// TIA Portal V17 export
// export: Created 2024-09-02T12:50:30.4708578Z, ExportSetting WithDefaults, DisplayName Totally Integrated Automation Portal, DisplayVersion V17, DisplayName TIA Portal Openness, DisplayVersion V17, DisplayName TIA Portal Version Control Interface, DisplayVersion V17, DisplayName STEP 7 Professional, DisplayVersion V17, DisplayName STEP 7 Safety, DisplayVersion V17, DisplayName WinCC Professional, DisplayVersion V17
TYPE "type_CognexVSin"
// stored: IsFailsafeCompliant false
   STRUCT
      Status : Struct
         Trigger_Ready : Bool;   // Aufnahmestatus: Trigger Ready / Recording status: Trigger Ready
         Trigger_Ack : Bool;   // Aufnahmestatus: Trigger Acknowledge / Recording status: Trigger Acknowledge
         Acquiring : Bool;   // Aufnahmestatus: Acquiring / Recording Status: Acquiring
         Missed_Ack : Bool;   // Aufnahmestatus: Missed Acknowledge / Recording Status: Missed Acknowledge
         Offline_Reason_0 : Bool;   // Aufnahmestatus: Offline Reason Bit 0 / Recording status: Offline Reason Bit 0
         Offline_Reason_1 : Bool;   // Aufnahmestatus: Offline Reason Bit 1 / Recording status: Offline Reason Bit 1
         Offline_Reason_2 : Bool;   // Aufnahmestatus: Offline Reason Bit 2 / Recording status: Offline Reason Bit 2
         Online : Bool;   // Aufnahmestatus: Online / Recording status: Online
         AcquisitionID_0 : Byte;   // Aufnahmestatus: Acquiring ID Bit 0 / Recording Status: Acquiring ID Bit 0
         AcquisitionID_1 : Byte;   // Aufnahmestatus: Acquiring ID Bit 1 / Recording Status: Acquiring ID Bit 1
         Inspecting : Bool;   // Inspektionsstatus: Inspecting / Inspection Status: Inspecting
         Inspection_complete : Bool;   // Inspektionsstatus: Inspection Complete / Inspection status: Inspection Complete
         Results_Buffer_Overrun : Bool;   // Inspektionsstatus: Results Buffer Overrung / Inspection Status: Results Buffer Overrung
         Results_valid : Bool;   // Inspektionsstatus: Results Valid / Inspection Status: Results Valid
         Job_loading : Bool;   // Inspektionsstatus: Job Loading / Inspection Status: Job Loading
         Job_load_complete : Bool;   // Inspektionsstatus: Job Load Complete / Inspection Status: Job Load Complete
         Job_load_failed : Bool;   // Inspektionsstatus: Job Load Failed / Inspection Status: Job Load Failed
         Res_37 : Bool;   // Inspektionsstatus: Reserve / Inspection status: Reserve
      END_STRUCT;
      Parameter : Struct
         Actual_Job_No : Byte;   // Parametersatz: Actual Job Number / Parameter set: Actual Job Number
         Res50 : Byte;
      END_STRUCT;
      Benutzerdaten : Struct
         Ausgabe : Array[0..3] of Byte;   // Systemausgaben / System diagnostic
         PID : Array[4..33] of Char;   // PID Reflektion / PID Reflection
         ProgNr_gueltig : Char;   // Programmnummer 1=gueltig / Program number 1=valid
         FehlerNr : Char;   // Fehlernummer 0=kein Fehler / Error number 0=no error
         Beleuchtungscheck : Char;   // Beleuchtungscheck 1=Beleuchtung IO / Lighting check 1=lighting IO
         ResSys : Array[37..42] of Char;   // Reserve
         Gesamtergebnis : Char;   // Gesamtergebnis / Overall result
         Teilergebnis_Code1 : Char;   // Teilergebnis 1 / Subtotal 1
         Codeguete_Code1 : Char;   // Codegüte 1 / Code quality 1
         Codeinhalt_Code1 : Array[46..103] of Char;   // Codeinhalt 1 / Code content 1
         Teilergebnis_Code2 : Char;   // Teilergebnis 2 / Subtotal 2
         Codeguete_Code2 : Char;   // Codegüte 2 / Code quality 2
         Codeinhalt_Code2 : Array[106..163] of Char;   // Codeinhalt 2 / Code content 2
         WeitereDaten : Array[164..221] of Char;   // Erweiterte Daten / Extended data
         Koordinate_X : DWord;   // X Koordinate / X Coordinate
         Koordinate_Y : DWord;   // Y Koordinate / X Coordinate
         Koordinate_Z : DWord;   // Z Koordinate / Z Coordinate
         Koordinate_A : DWord;   // Winkel Koordinate / Angle Coordinate
         Reserve : Array[238..253] of Char;   // Reserve
      END_STRUCT;
   END_STRUCT;
END_TYPE
